PROGRAM Axis1_Motion
VAR
	//power
	MC_Power_Axis1: MC_Power;
	//Move
	m_State_Axis1: INT;
	MC_MoveAbsolute_Axis1: MC_MoveAbsolute;

	//JOG
	j_State_Axis1: INT;
	MC_JOG_Axis1: MC_Jog;

	//Stop
	MC_Stop_Axis1: MC_Stop;
	s_State_Axis1: INT;

	//reset
	r_State_Axis1: INT;
	MC_Reset_Axis1: MC_Reset;

	//setposition
	MC_SetPosition_Axis1: MC_SetPosition;
	sp_State_Axis1: INT;
	SetPosition_delay_Axis1:TON;

	//button interlock
	Axis1_J1: BOOL;//JOG+
	Axis1_J2: BOOL;//JOG-
	Axis1_P: BOOL;//Position moving
	Axis1_S: BOOL;//Stop
	Axis1_SP: BOOL;//set position
	//input protect
	Axis1_PositionProtectionSet:BOOL;
	Axis1_InputPositionOutOfRange:BOOL;
	es_State_Axis1: INT;
	FTrig_ReachLS1: F_TRIG;
	RTrig_EStop1:R_TRIG;
	btn_ReachLSReset_Axis1: BOOL;
END_VAR

//
//输入保护
//
IF btn_Move_Axis1 THEN
	IF targetPositionAxis1>=Axis1_minPosition AND targetPositionAxis1<=Axis1_maxPosition THEN
		Axis1_InputPositionOutOfRange:=FALSE;
		Error:=FALSE;
		ErrorId:=0;
		ErrorDescription:='';
	ELSE
		Axis1_InputPositionOutOfRange:=TRUE;
		Error:=TRUE;
		ErrorId:=1001;
		ErrorDescription:='Axis1_InputPositionOutOfRange';
		RETURN;
	END_IF
END_IF
IF btn_JogForward_Axis1 THEN
	IF Axis1_CurrentPosition_retain+increaseJogPositionAxis1<=Axis1_maxPosition  THEN
		Axis1_InputPositionOutOfRange:=FALSE;
		Error:=FALSE;
		ErrorId:=0;
		ErrorDescription:='';
	ELSE
		Axis1_InputPositionOutOfRange:=TRUE;
		Error:=TRUE;
		ErrorId:=1002;
		ErrorDescription:='exceed Axis1_maxPosition';
		RETURN;
	END_IF
END_IF 

IF  btn_JogBackward_Axis1 THEN
	IF Axis1_CurrentPosition_retain-increaseJogPositionAxis1>=Axis1_minPosition  THEN
		Axis1_InputPositionOutOfRange:=FALSE;
		Error:=FALSE;
		ErrorId:=0;
		ErrorDescription:='';
	ELSE
		Axis1_InputPositionOutOfRange:=TRUE;
		Error:=TRUE;
		ErrorId:=1003;
		ErrorDescription:='less than Axis1_minPosition';
		RETURN;
	END_IF
END_IF
//
//运行状态指示
//
Axis1.ReadStatus();
IF  Axis1.Status.Moving  THEN
	Axis1_moving:=TRUE;
ELSE
	Axis1_moving:=FALSE;
END_IF;
//
//电机错误指示
//
IF  axis1.NcToPlc.ErrorCode=0 THEN
	Axis1_error     := FALSE;
ELSE
	Axis1_error     := TRUE;
	Error:=TRUE;
	ErrorId:=1002;
	ErrorDescription:='axis1.NcToPlc.ErrorCode=0';
END_IF;
//
//Moving_done_Axis1
//
//
Moving_done_Axis1:=MC_MoveAbsolute_Axis1.Done OR MC_JOG_Axis1.Done;
//
//Positioning move
//
A_MCAxis1();
CASE m_State_Axis1 OF 
	0:
		//检查是否有错误等
		IF  NOT Axis1_error THEN
			m_State_Axis1:=1;
		ELSE
			m_State_Axis1:=-100;
		END_IF
	1:
		//检查电机是否已经上电，如无，则上电
		IF 	NOT MC_Power_Axis1.Status THEN
			MC_Power_Axis1.Enable:=TRUE;
		ELSE
			m_State_Axis1:=2;
		END_IF
	2:
		//定位运行
		MC_MoveAbsolute_Axis1.Position:=targetPositionAxis1;
		MC_MoveAbsolute_Axis1.Velocity:=targetVelocityAxis1;
		IF btn_Move_Axis1 THEN
			MC_MoveAbsolute_Axis1.Execute:=TRUE;
			m_State_Axis1:=3;
		END_IF
	3:
		//是否运动到位
		IF MC_MoveAbsolute_Axis1.Done THEN
			m_State_Axis1:=88;
		END_IF
	88:
		btn_Move_Axis1:=FALSE;
		MC_MoveAbsolute_Axis1.Execute:=FALSE;
		m_State_Axis1:=0;		
	-100:
		btn_Move_Axis1:=FALSE;
		MC_MoveAbsolute_Axis1.Execute:=FALSE;
		Error:=TRUE;
		Axis1_error:=TRUE;
		ErrorId:=1002;
		ErrorDescription:='E_STOP AND NOT Axis1_error';
		
END_CASE
//
//JOG+
//
CASE j_State_Axis1 OF 
	0:
		//检查是否有错误等
		IF  NOT Axis1_error THEN
			j_State_Axis1:=1;
		ELSE
			j_State_Axis1:=-100;
		END_IF
	1:
		//检查电机是否已经上电，如无，则上电
		IF 	NOT MC_Power_Axis1.Status THEN
			MC_Power_Axis1.Enable:=TRUE;
		ELSE
			j_State_Axis1:=2;
		END_IF
	2:
		//JOG运行
		MC_JOG_Axis1.Position:=increaseJogPositionAxis1;
		MC_JOG_Axis1.Velocity:=targetVelocityAxis1;
		IF btn_JogForward_Axis1 AND NOT btn_JogBackward_Axis1 THEN
			MC_JOG_Axis1.JogForward:=TRUE;
			j_State_Axis1:=3;
		END_IF
		IF btn_JogBackward_Axis1 AND NOT btn_JogForward_Axis1 THEN
			MC_JOG_Axis1.JogBackwards:=TRUE;
			j_State_Axis1:=3;
		END_IF
	3:
		//是否运动到位
		IF btn_JogForward_Axis1 THEN
			btn_JogForward_Axis1:=FALSE;
		END_IF 
		IF btn_JogBackward_Axis1 THEN
			btn_JogBackward_Axis1:=FALSE;
		END_IF
		IF MC_JOG_Axis1.Done THEN
			j_State_Axis1:=88;
		END_IF
	88:
		MC_JOG_Axis1.JogForward:=FALSE;
		MC_JOG_Axis1.JogBackwards:=FALSE;
		btn_JogForward_Axis1:=FALSE;
		btn_JogBackward_Axis1:=FALSE;
		j_State_Axis1:=0;	
		
	-100:
		MC_JOG_Axis1.JogForward:=FALSE;
		MC_JOG_Axis1.JogBackwards:=FALSE;
		btn_JogForward_Axis1:=FALSE;
		btn_JogBackward_Axis1:=FALSE;
		Error:=TRUE;
		Axis1_error:=TRUE;
		ErrorId:=1002;
		ErrorDescription:='E_STOP AND NOT Axis1_error';	
END_CASE
//
//STOP
//
CASE s_State_Axis1 OF 
	0:
		s_State_Axis1:=1;
	1:
		//检查电机是否已经上电，如无，则上电
		IF 	NOT MC_Power_Axis1.Status THEN
			MC_Power_Axis1.Enable:=TRUE;
		ELSE
			s_State_Axis1:=2;
		END_IF
	2:
		//STOP
		IF btn_Stop_Axis1 THEN
			MC_Stop_Axis1.Execute:=TRUE;
			s_State_Axis1:=3;
		END_IF
	3:
		//是否运动到位
		IF MC_Stop_Axis1.Done THEN
			s_State_Axis1:=88;
		END_IF
	88:
		btn_Stop_Axis1:=FALSE;
		MC_Stop_Axis1.Execute:=FALSE;
		s_State_Axis1:=0;	
		//reset status
		btn_Move_Axis1:=FALSE;
		MC_MoveAbsolute_Axis1.Execute:=FALSE;
		btn_JogForward_Axis1:=FALSE;
		btn_JogBackward_Axis1:=FALSE;
		MC_JOG_Axis1.JogForward:=FALSE;
		MC_JOG_Axis1.JogBackwards:=FALSE;
		m_State_Axis1:=0;
		j_State_Axis1:=0;
	-100:
		btn_Stop_Axis1:=FALSE;
		MC_Stop_Axis1.Execute:=FALSE;
		Error:=TRUE;
		Axis1_error:=TRUE;
		ErrorId:=1002;
		ErrorDescription:='E_STOP AND NOT Axis1_error';
		//reset status
		btn_Move_Axis1:=FALSE;
		MC_MoveAbsolute_Axis1.Execute:=FALSE;
		btn_JogForward_Axis1:=FALSE;
		btn_JogBackward_Axis1:=FALSE;
		MC_JOG_Axis1.JogForward:=FALSE;
		MC_JOG_Axis1.JogBackwards:=FALSE;
		m_State_Axis1:=0;
		j_State_Axis1:=0;
END_CASE
//
//Reset
//
CASE r_State_Axis1 OF 
	0:
		IF btn_Reset_Axis1 OR btn_ReachLSReset_Axis1 THEN
			MC_Reset_Axis1.Execute:=TRUE;
			r_State_Axis1:=1;
		END_IF
	1:
		//是否运动到位
		IF MC_Reset_Axis1.Done THEN
			r_State_Axis1:=88;
		END_IF
	88:
		r_State_Axis1:=0;
		MC_Reset_Axis1.Execute:=FALSE;	
		btn_Reset_Axis1:=FALSE;
		btn_ReachLSReset_Axis1:=FALSE;
		//reset status
		btn_Move_Axis1:=FALSE;
		MC_MoveAbsolute_Axis1.Execute:=FALSE;
		btn_JogForward_Axis1:=FALSE;
		btn_JogBackward_Axis1:=FALSE;
		MC_JOG_Axis1.JogForward:=FALSE;
		MC_JOG_Axis1.JogBackwards:=FALSE;
		m_State_Axis1:=0;
		s_State_Axis1:=0;
		j_State_Axis1:=0;
END_CASE
//
//setposotion
//
SetPosition_delay_Axis1.PT:=T#0.1S;
SetPosition_delay_Axis1();
IF btn_SetPosition_Axis1 THEN
	CASE sp_State_Axis1 OF 
		0:
			IF NOT Axis1_moving THEN
				sp_State_Axis1:=1;
			END_IF
		1:
			MC_SetPosition_Axis1.Position:=PositionSetValue_Axis1;
			MC_SetPosition_Axis1.Execute:=TRUE;
			SetPosition_delay_Axis1.IN:=TRUE;
			sp_State_Axis1:=2;
		2:
			IF MC_SetPosition_Axis1.Done THEN
				sp_State_Axis1:=88;
			END_IF
			IF SetPosition_delay_Axis1.Q THEN//延时结束时，还没有设置位置成功
				sp_State_Axis1:=-100;
			END_IF
		88:
			PositionSetDone_Axis1:=TRUE;
			MC_SetPosition_Axis1.Execute:=FALSE;
			SetPosition_delay_Axis1.IN:=FALSE;
			sp_State_Axis1:=0;
			btn_SetPosition_Axis1:=FALSE;
		-100:
			PositionSetDone_Axis1:=FALSE;
			MC_SetPosition_Axis1.Execute:=FALSE;
			SetPosition_delay_Axis1.IN:=FALSE;
			btn_SetPosition_Axis1:=FALSE;
	END_CASE
END_IF
//
//
//
//急停
IF NOT(E_STOP AND E_STOP_rem AND Plc_EmergencyStop) THEN
	CASE es_State_Axis1 OF
		0:
			es_State_Axis1:=1;
		1:
			E_STOP_led:= FALSE;	//red
			MC_Power_Axis1.Enable:=FALSE;//电机2断电
			btn_Stop_Axis1:=TRUE;//STOP axis1
			A_MCAxis1();
			Error:=TRUE;
			ErrorId:=101;
			ErrorDescription:='E_STOP';
	END_CASE
END_IF

RTrig_EStop1(CLK:=E_STOP AND E_STOP_rem AND Plc_EmergencyStop);
IF RTrig_EStop1.Q THEN
	E_STOP_led:= TRUE;	//green
	Error:=FALSE;
	ErrorId:=0;
	ErrorDescription:='';
END_IF

(*触发限位开关后，相当于点击了Stop按钮*)
FTrig_ReachLS1(CLK:=foreward_limit_axis1 AND backward_limit_axis1);
IF FTrig_ReachLS1.Q THEN
	btn_Reset_Axis1:=TRUE;
	btn_ReachLSReset_Axis1:=TRUE;
END_IF


//
//屏幕按钮**互锁变量,FALSE时，该按钮灰色不能触发
//
//J1->JOG+
IF  foreward_limit_axis1 AND E_STOP  AND Local_led AND NOT  Axis1_error  AND NOT  Axis1_moving AND
	NOT btn_Move_Axis1 AND NOT  btn_JogBackward_Axis1  THEN
	Axis1_J1     := TRUE;
ELSE
	Axis1_J1     := FALSE;
END_IF;
//J2>JOG-
IF  backward_limit_axis1  AND E_STOP   AND Local_led AND NOT  Axis1_error  AND NOT  Axis1_moving AND 
	 NOT  btn_Move_Axis1 AND NOT btn_JogForward_Axis1 THEN
	Axis1_J2     := TRUE;
ELSE
	Axis1_J2     := FALSE;
END_IF;
//P->PositionMove
IF  E_STOP   AND Local_led AND NOT  Axis1_error  AND NOT  Axis1_moving AND 
	 NOT btn_JogForward_Axis1  AND NOT  btn_JogBackward_Axis1 THEN
	Axis1_P     := TRUE;
ELSE
	Axis1_P     := FALSE;
END_IF;
//SP->SetPosition
IF E_STOP  AND Local_led AND NOT  Axis1_error  AND NOT Axis1_moving  THEN
	Axis1_SP     := TRUE;
ELSE
	Axis1_SP     := FALSE;
END_IF;
//S->Stop
IF E_STOP  AND Local_led AND NOT  Axis1_error THEN
	Axis1_S     := TRUE;
ELSE
	Axis1_S     := FALSE;
END_IF;

ACTION A_MCAxis1:
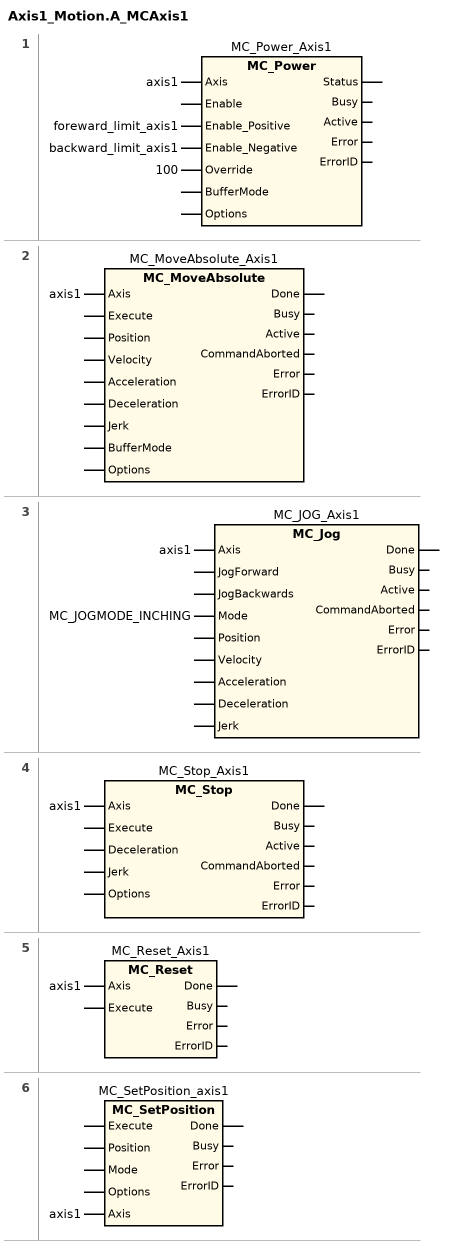
// NETWORK 1
MC_Power_Axis1(
    Axis := axis1,
    Enable_Positive := foreward_limit_axis1,
    Enable_Negative := backward_limit_axis1,
    Override := 100); // MC_Power

// NETWORK 2
MC_MoveAbsolute_Axis1(Axis := axis1); // MC_MoveAbsolute

// NETWORK 3
MC_JOG_Axis1(Axis := axis1, Mode := MC_JOGMODE_INCHING); // MC_Jog

// NETWORK 4
MC_Stop_Axis1(Axis := axis1); // MC_Stop

// NETWORK 5
MC_Reset_Axis1(Axis := axis1); // MC_Reset

// NETWORK 6
MC_SetPosition_axis1(Axis := axis1); // MC_SetPosition
END_ACTION

END_PROGRAM

(* stored: Version 1.1.0.1, ProductVersion 3.1.4024.6
   POU Axis1_Motion: Id {bfe68869-bf5b-4e26-9fd3-de7a537cc7f6}, SpecialFunc None
   Action A_MCAxis1: Id {10c0b877-c729-48f5-a9bd-16c8e6afc448} *)
